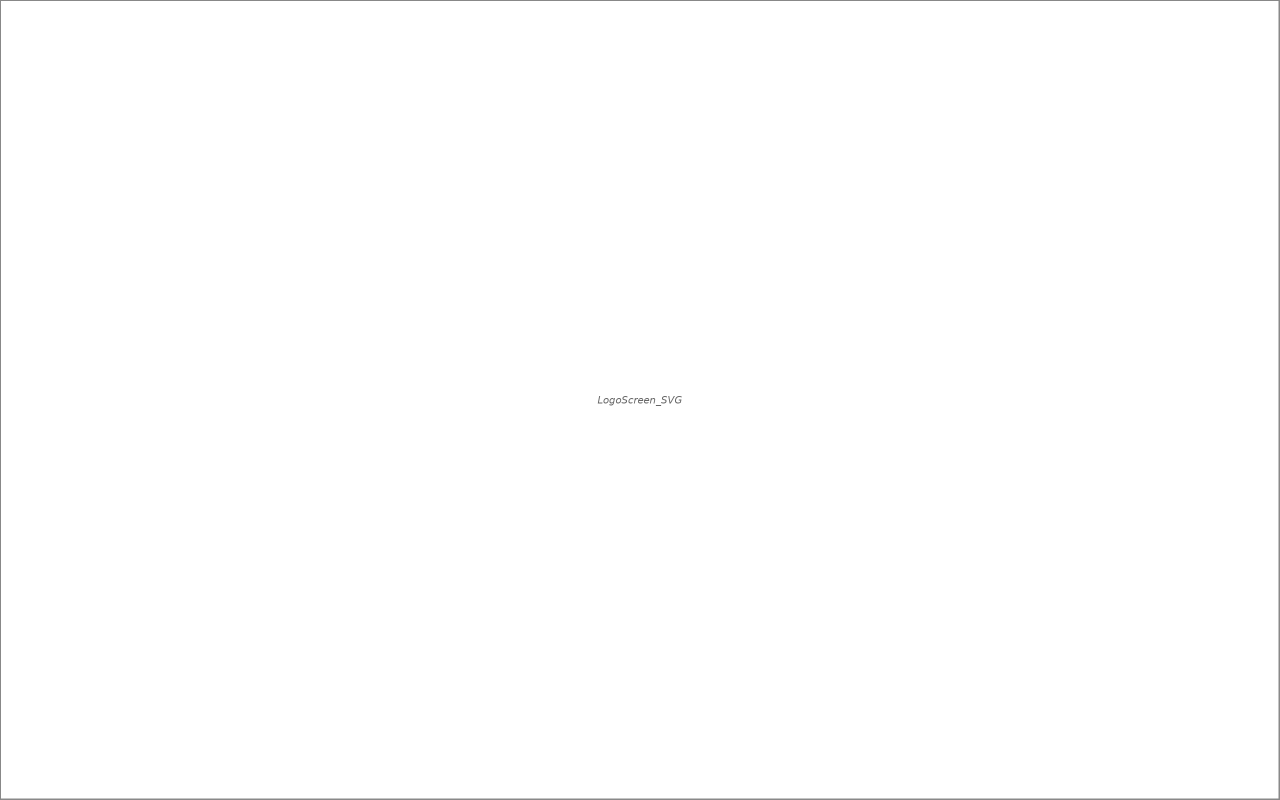
VISUALIZATION Idle  // 1280x800
VAR_IN_OUT
	nUnitsProduced : UDINT ; // Units produced in machine lifetime
END_VAR
    Frame (0,0 1280x800), frame switch variable: 0
        shows LogoScreen_SVG(nUnitsProduced := nUnitsProduced)
        shows Settings()
        shows ParameterScreen()
        shows Run()
END_VISUALIZATION

(* stored: Version 1.1.0.1, ProductVersion 3.1.4024.5
   Visu Idle: Id {9c0dfbb2-ead7-41c1-9ffd-e66a861a7940} *)
